PROGRAM MAIN
VAR
	_testContext : TcoBlinkerTestContext;
	_testEvalueateMeasurementContext : TcoEvaluateMeasurementContext;
END_VAR

_testContext.ProbeRun();
_testEvalueateMeasurementContext.ProbeRun();

END_PROGRAM

(* stored: Version 1.1.0.1, ProductVersion 3.1.4024.10
   POU MAIN: Id {6af77bf1-277e-0a98-2c35-6eb9f887cb1b}, SpecialFunc None *)
